% RSLogix 500 project Project2.RSS, saved by version 8.30.00.16 %
PROJECT "2"    % processor: Bul.1763 MicroLogix 1100 Series B %

PROGRAM FILES
  LAD 2 "MAIN"  3 rungs
  LAD 3 "I/0"  8 rungs
  LAD 4 "CONTROLS"  8 rungs

DATA FILES
  O0 OUTPUT  4 elements
  I1 INPUT  6 elements
  S2 STATUS  66 elements
  B3 BINARY  2 elements
  T4 TIMER  1 elements
  C5 COUNTER  1 elements
  R6 CONTROL  1 elements
  N7 INTEGER  1 elements
  F8 FLOAT  1 elements

LADDER 2 "MAIN"
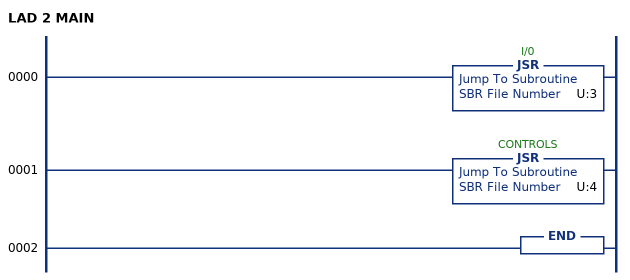
% Rung: 0 %
SOR JSR U:3 EOR
%   U:3  "I/0" %
% Rung: 1 %
SOR JSR U:4 EOR
%   U:4  "CONTROLS" %
% Rung: 2 %
SOR END EOR

LADDER 3 "I/0"
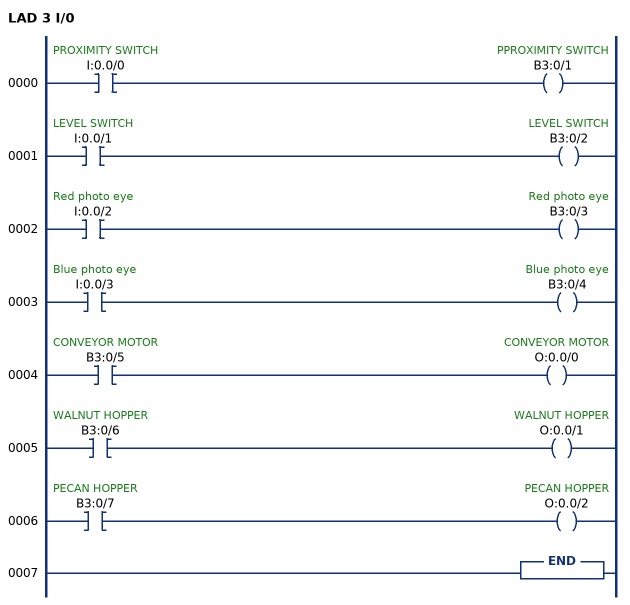
% Rung: 0 %
SOR XIC I:0.0/0 OTE B3:0/1 EOR
%   I:0.0/0  "PROXIMITY SWITCH" %
%   B3:0/1  "PPROXIMITY SWITCH" %
% Rung: 1 %
SOR XIC I:0.0/1 OTE B3:0/2 EOR
%   I:0.0/1  "LEVEL SWITCH" %
%   B3:0/2  "LEVEL SWITCH" %
% Rung: 2 %
SOR XIC I:0.0/2 OTE B3:0/3 EOR
%   I:0.0/2  "Red photo eye" %
%   B3:0/3  "Red photo eye" %
% Rung: 3 %
SOR XIC I:0.0/3 OTE B3:0/4 EOR
%   I:0.0/3  "Blue photo eye" %
%   B3:0/4  "Blue photo eye" %
% Rung: 4 %
SOR XIC B3:0/5 OTE O:0.0/0 EOR
%   B3:0/5  "CONVEYOR MOTOR" %
%   O:0.0/0  "CONVEYOR MOTOR" %
% Rung: 5 %
SOR XIC B3:0/6 OTE O:0.0/1 EOR
%   B3:0/6  "WALNUT HOPPER" %
%   O:0.0/1  "WALNUT HOPPER" %
% Rung: 6 %
SOR XIC B3:0/7 OTE O:0.0/2 EOR
%   B3:0/7  "PECAN HOPPER" %
%   O:0.0/2  "PECAN HOPPER" %
% Rung: 7 %
SOR END EOR

LADDER 4 "CONTROLS"
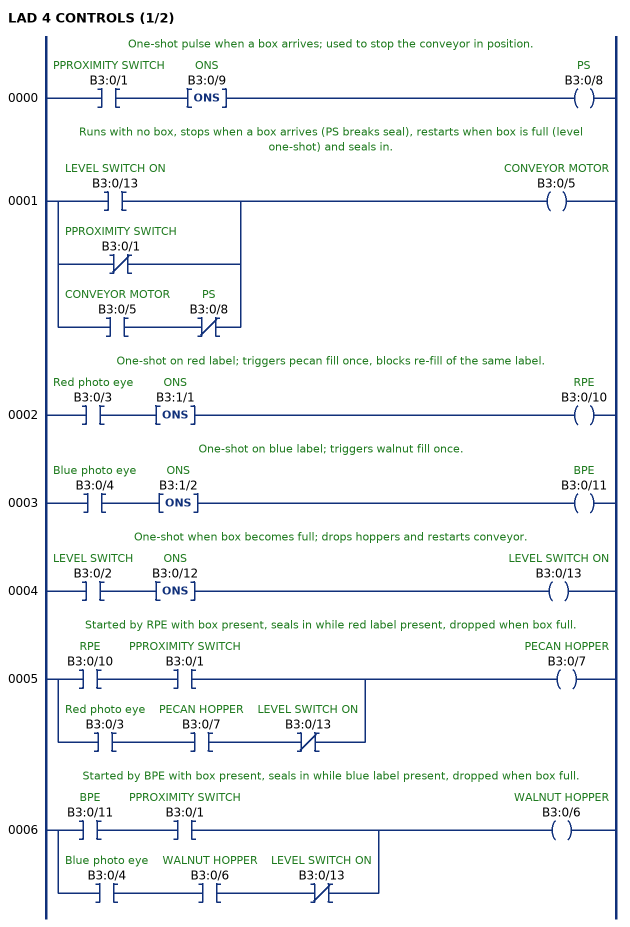
% Rung: 0 %
% One-shot pulse when a box arrives; used to stop the conveyor in position. %
SOR XIC B3:0/1 ONS B3:0/9 OTE B3:0/8 EOR
%   B3:0/1  "PPROXIMITY SWITCH" %
%   B3:0/9  "ONS" %
%   B3:0/8  "PS" %
% Rung: 1 %
% Runs with no box, stops when a box arrives (PS breaks seal), restarts when box is full (level one-shot) and seals in. %
SOR BST BST XIC B3:0/13 NXB XIO B3:0/1 BND NXB XIC B3:0/5 XIO B3:0/8 BND OTE B3:0/5 EOR
%   B3:0/13  "LEVEL SWITCH ON" %
%   B3:0/1  "PPROXIMITY SWITCH" %
%   B3:0/5  "CONVEYOR MOTOR" %
%   B3:0/8  "PS" %
% Rung: 2 %
% One-shot on red label; triggers pecan fill once, blocks re-fill of the same label. %
SOR XIC B3:0/3 ONS B3:1/1 OTE B3:0/10 EOR
%   B3:0/3  "Red photo eye" %
%   B3:1/1  "ONS" %
%   B3:0/10  "RPE" %
% Rung: 3 %
% One-shot on blue label; triggers walnut fill once. %
SOR XIC B3:0/4 ONS B3:1/2 OTE B3:0/11 EOR
%   B3:0/4  "Blue photo eye" %
%   B3:1/2  "ONS" %
%   B3:0/11  "BPE" %
% Rung: 4 %
% One-shot when box becomes full; drops hoppers and restarts conveyor. %
SOR XIC B3:0/2 ONS B3:0/12 OTE B3:0/13 EOR
%   B3:0/2  "LEVEL SWITCH" %
%   B3:0/12  "ONS" %
%   B3:0/13  "LEVEL SWITCH ON" %
% Rung: 5 %
% Started by RPE with box present, seals in while red label present, dropped when box full. %
SOR BST XIC B3:0/10 XIC B3:0/1 NXB XIC B3:0/3 XIC B3:0/7 XIO B3:0/13 BND OTE B3:0/7 EOR
%   B3:0/10  "RPE" %
%   B3:0/1  "PPROXIMITY SWITCH" %
%   B3:0/3  "Red photo eye" %
%   B3:0/7  "PECAN HOPPER" %
%   B3:0/13  "LEVEL SWITCH ON" %
% Rung: 6 %
% Started by BPE with box present, seals in while blue label present, dropped when box full. %
SOR BST XIC B3:0/11 XIC B3:0/1 NXB XIC B3:0/4 XIC B3:0/6 XIO B3:0/13 BND OTE B3:0/6 EOR
%   B3:0/11  "BPE" %
%   B3:0/1  "PPROXIMITY SWITCH" %
%   B3:0/4  "Blue photo eye" %
%   B3:0/6  "WALNUT HOPPER" %
%   B3:0/13  "LEVEL SWITCH ON" %

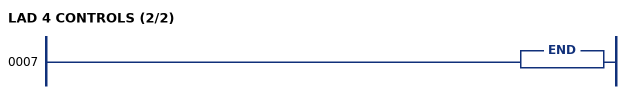
% Rung: 7 %
SOR END EOR

COMMENTS NOT ATTACHED TO A CURRENT RUNG
  B3:0/5: Runs with no box, stops when a box arrives (PS breaks seal), restarts when box is full (level one-shot) and seals in.

REVISION NOTES
  0: VERSION2
  1: VERSION 1
  2: VERSION3
  3: VERSION4
  4: FINAL VERSION
  5: CHECKING VERVISION5
  6: CHECKING VERSION 6
  7: CHECKING VERSION 7
  8: VERSION9
  9: FINAL VERSION
  10: with comments
